// TIA Portal V20 export
TYPE "typeSequenceControlNodeJobInterfaceCommands"
// stored: Namespace Unit1.Em2
   STRUCT
      reqEm0Rewind { ExternalWritable := 'False'} : Bool;
      reqEm1Rewind { ExternalWritable := 'False'} : Bool;
      reqEm0To1LinkChg { ExternalWritable := 'False'} : Bool;
      reqEm1To0LinkChg { ExternalWritable := 'False'} : Bool;
   END_STRUCT;
END_TYPE
